// TIA Portal V18 export
// export: Created 2025-12-01T17:50:25.6597792Z, ExportSetting None, DisplayName Totally Integrated Automation Portal, DisplayVersion V18 Update 5, DisplayName TIA Portal Openness, DisplayVersion V18 Update 5, DisplayName TIA Portal Teamcenter Gateway, DisplayVersion V18, DisplayName TIA Portal Version Control Interface, DisplayVersion V18, DisplayName STEP 7 Professional, DisplayVersion V18 Update 5, DisplayName STEP 7 Safety, DisplayVersion V18, DisplayName WinCC Professional, DisplayVersion V18 Update 5
ORGANIZATION_BLOCK "08_HW_INT0"   // OB40, LAD, HardwareInterrupt
TITLE = "Hardware Interrupt"
{ S7_Optimized_Access := 'FALSE' }
// stored: AutoNumber false, SetENOAutomatically false
   VAR_TEMP
      OB40_EV_CLASS : Byte;   // Bits 0-3 = 1 (Coming event), Bits 4-7 = 1 (Event class 1)
      OB40_STRT_INF : Byte;   // 16#41 (OB 40 has started)
      OB40_PRIORITY : Byte;   // Priority of OB Execution
      OB40_OB_NUMBR : Byte;   // 40 (Organization block 40, OB40)
      OB40_RESERVED_1 : Byte;   // Reserved for system
      OB40_IO_FLAG : Byte;   // 16#54 (input module), 16#55 (output module)
      OB40_MDL_ADDR : Word;   // Base address of module initiating interrupt
      OB40_POINT_ADDR : DWord;   // Interrupt status of the module
      OB40_DATE_TIME : Date_And_Time;   // Date and time OB40 started
   END_VAR
BEGIN
END_ORGANIZATION_BLOCK
